// TIA Portal project "Project_asynchronousmotor_startdeltastarting" (V16)

(* hardware
DEVICE "S7-1200 station_1"  S7-1200 Station
   slot 0: "Rack_0"  S7-1200 Rack  Rack  V1.0
   slot 1: "PLC_1"  CPU 1212C DC/DC/Rly  6ES7 212-1HE40-0XB0  V4.4
   slot 2: "DQ 8x24VDC _1"  SM 1222 DQ8 x 24VDC  6ES7 222-1BF32-0XB0  V2.0
   slot 3: "DI 4x24VDC_1"  DI4 signal board (200 kHz)  6ES7 221-3BD30-0XB0  V1.0
*)

// ===== PLC "PLC_1"  CPU 1212C DC/DC/Rly =====

VAR_GLOBAL   // PLC tag table "Default tag table"
   "START BUT" AT %I4.0 : Bool;
   "STOP BUT" AT %I4.1 : Bool;
   "ANA KONT" AT %Q8.0 : Bool;
   "YILDIZ KONT" AT %Q8.1 : Bool;
   "UCGEN KONT" AT %Q8.2 : Bool;
END_VAR

// folder: System blocks/Program resources

DATA_BLOCK "TIMER 1"   // DB1
{ S7_Optimized_Access := 'TRUE' }
AUTHOR : Simatic
FAMILY : IEC
NAME : IEC_TMR
VERSION : 1.0
// stored: InstanceOfName IEC_TIMER
"IEC_TIMER"
BEGIN
END_DATA_BLOCK

// folder: (top level)

ORGANIZATION_BLOCK "Main"   // OB1, LAD, ProgramCycle
TITLE = "Main Program Sweep (Cycle)"
{ S7_Optimized_Access := 'TRUE' }
VERSION : 0.1
   VAR_INPUT
      Initial_Call : Bool;   // Initial call of this OB
      Remanence : Bool;   // =True, if remanent data are available
   END_VAR
BEGIN

REGION Network 1: SİSTEMİN BESLEMESİ
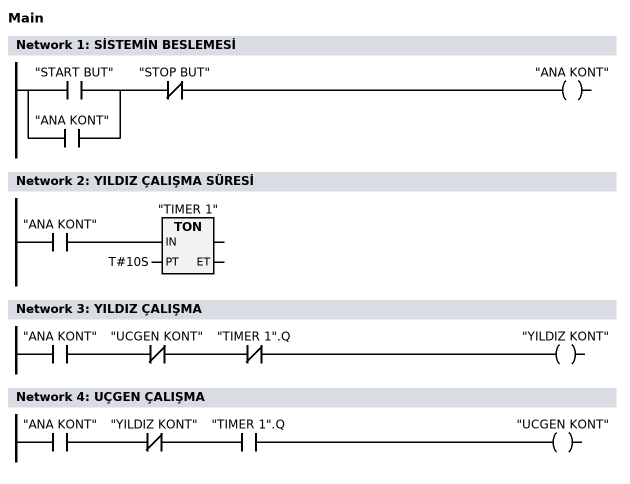
   RUNG wire#powerrail
      Contact( "START BUT" )
      wire#w1
      I_Contact( "STOP BUT" )
      Coil( "ANA KONT" )
   END_RUNG
   RUNG wire#powerrail
      Contact( "ANA KONT" )
   END_RUNG wire#w1
   // the same network as SCL:
   "ANA KONT" := ("START BUT" OR "ANA KONT") AND NOT "STOP BUT";
END_REGION

REGION Network 2: YILDIZ ÇALIŞMA SÜRESİ
   "TIMER 1".TON(IN := "ANA KONT", PT := T#10S);
END_REGION

REGION Network 3: YILDIZ ÇALIŞMA
   RUNG wire#powerrail
      Contact( "ANA KONT" )
      I_Contact( "UCGEN KONT" )
      I_Contact( "TIMER 1".Q )
      Coil( "YILDIZ KONT" )
   END_RUNG
   // the same network as SCL:
   "YILDIZ KONT" := "ANA KONT" AND NOT "UCGEN KONT" AND NOT "TIMER 1".Q;
END_REGION

REGION Network 4: UÇGEN ÇALIŞMA
   RUNG wire#powerrail
      Contact( "ANA KONT" )
      I_Contact( "YILDIZ KONT" )
      Contact( "TIMER 1".Q )
      Coil( "UCGEN KONT" )
   END_RUNG
   // the same network as SCL:
   "UCGEN KONT" := "ANA KONT" AND NOT "YILDIZ KONT" AND "TIMER 1".Q;
END_REGION
END_ORGANIZATION_BLOCK